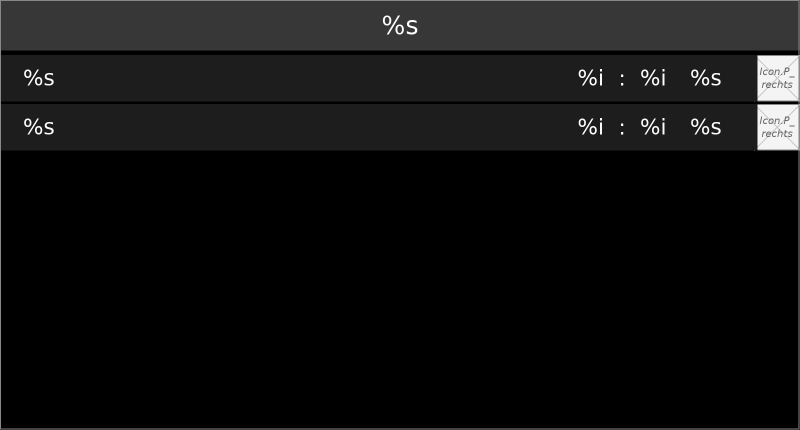
VISUALIZATION CLK_D_Tagesprogramm_Liste  // 800x430
VAR_IN_OUT
	FB_CLK_D:CLK_D;
	
END_VAR
VAR_INPUT
	i_Titel:INT;
END_VAR
	
VAR

	
	
END_VAR
    Rectangle (0,425 800x5)
    Rectangle (0,0 800x50), "%s", text list: 'Sprachen', text index: i_Titel
    Rectangle (0,55 800x46)
    Rectangle (20,55 400x46), "%s", text list: 'Sprachen', text index: 93
    Image (754,55 46x46), image: Icon.P_rechts
        OnMouseClick: execute { Visu.i_Frame_Index:=1; }
    Rectangle (637,55 49x46), "%i", text variable: FB_CLK_D.t_Ein.wMinute
    Rectangle (537,55 70x46), "%i", text variable: FB_CLK_D.t_Ein.wHour
    Rectangle (617,55 10x46), ":"
    Rectangle (687,55 70x46), "%s", text list: 'Sprachen', text index: 74
    Rectangle (0,104 800x46)
    Rectangle (20,104 400x46), "%s", text list: 'Sprachen', text index: 94
    Image (754,104 46x46), image: Icon.P_rechts
        OnMouseClick: execute { Visu.i_Frame_Index:=2; }
    Rectangle (637,104 49x46), "%i", text variable: FB_CLK_D.t_Aus.wMinute
    Rectangle (537,104 70x46), "%i", text variable: FB_CLK_D.t_Aus.wHour
    Rectangle (617,104 10x46), ":"
    Rectangle (687,104 70x46), "%s", text list: 'Sprachen', text index: 74
END_VISUALIZATION

// ZY_Visu/Zeitprogramm/CLK_I/CLK_I_Tagesimpuls
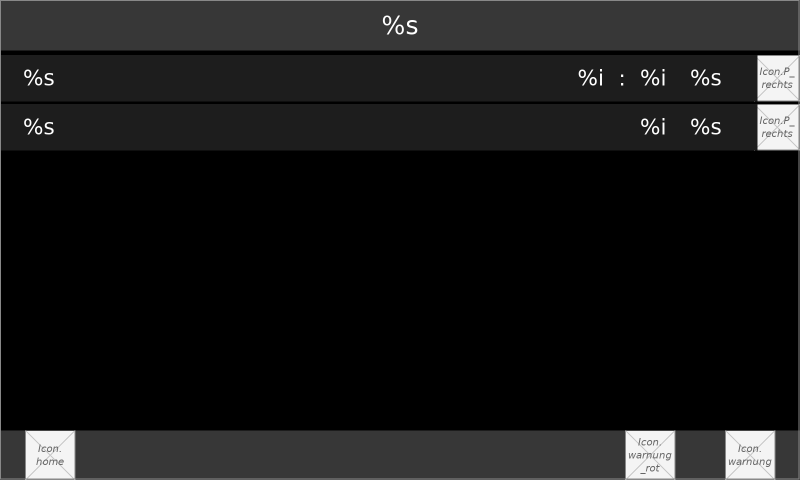
VISUALIZATION CLK_I_Tagesimpuls  // 800x480
VAR_IN_OUT
	FB_CLK_I:CLK_I;

END_VAR
    Frame (0,430 800x50)
        shows Fusszeile_50()
    Frame (0,0 800x430), frame switch variable: Visu.i_Frame_Index
        shows CLK_I_Tagesimpuls_Liste(i_Titel := 76, FB_CLK_I := FB_CLK_I)
        shows Ein_Aus_Zeit_aendern(i_titel := 68, i_Minuten := FB_CLK_I.t_Ein.wMinute, i_Stunden := FB_CLK_I.t_Ein.wHour)
        shows Sekunden_aendern(i_titel := 102, i_Sekunden := FB_CLK_I.t_Imp.wSecond)
END_VISUALIZATION

// ZY_Visu/Zeitprogramm/CLK_I/CLK_I_Tagesimpuls_Liste
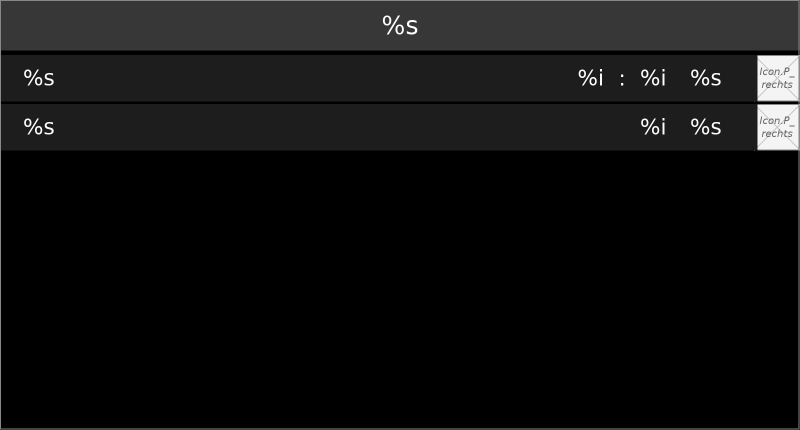
VISUALIZATION CLK_I_Tagesimpuls_Liste  // 800x430
VAR_IN_OUT
	FB_CLK_I:CLK_I;
	
END_VAR
VAR_INPUT
	i_Titel:INT;
END_VAR
	
VAR

	
	
END_VAR
    Rectangle (0,425 800x5)
    Rectangle (0,0 800x50), "%s", text list: 'Sprachen', text index: i_Titel
    Rectangle (0,55 800x46)
    Rectangle (20,55 400x46), "%s", text list: 'Sprachen', text index: 93
    Image (754,55 46x46), image: Icon.P_rechts
        OnMouseClick: execute { Visu.i_Frame_Index:=1; }
    Rectangle (637,55 49x46), "%i", text variable: FB_CLK_I.t_Ein.wMinute
    Rectangle (537,55 70x46), "%i", text variable: FB_CLK_I.t_Ein.wHour
    Rectangle (617,55 10x46), ":"
    Rectangle (687,55 70x46), "%s", text list: 'Sprachen', text index: 74
    Rectangle (0,104 800x46)
    Rectangle (20,104 400x46), "%s", text list: 'Sprachen', text index: 102
    Image (754,104 46x46), image: Icon.P_rechts
        OnMouseClick: execute { Visu.i_Frame_Index:=2; }
    Rectangle (637,104 49x46), "%i", text variable: FB_CLK_I.t_Imp.wSecond
    Rectangle (687,104 70x46), "%s", text list: 'Sprachen', text index: 103
END_VISUALIZATION

// ZY_Visu/Zeitprogramm/CLK_M/CLK_M_Monatsimpuls
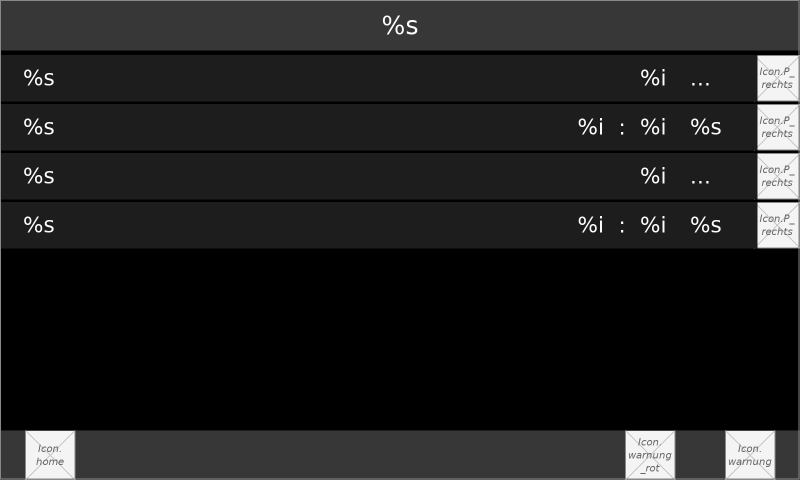
VISUALIZATION CLK_M_Monatsimpuls  // 800x480
VAR_IN_OUT
	FB_CLK_M:CLK_M;

END_VAR
    Frame (0,430 800x50)
        shows Fusszeile_50()
    Frame (0,0 800x430), frame switch variable: Visu.i_Frame_Index
        shows CLK_M_Monatsimpuls_Liste(i_Titel := 78, FB_CLK_M := FB_CLK_M)
        shows Monatstag_aendern(i_titel := 99, i_Monatstag := FB_CLK_M.t_Ein.wDay)
        shows Ein_Aus_Zeit_aendern(i_titel := 68, i_Minuten := FB_CLK_M.t_Ein.wMinute, i_Stunden := FB_CLK_M.t_Ein.wHour)
        shows Monatstag_aendern(i_titel := 99, i_Monatstag := FB_CLK_M.t_Aus.wDay)
        shows Ein_Aus_Zeit_aendern(i_titel := 68, i_Minuten := FB_CLK_M.t_Aus.wMinute, i_Stunden := FB_CLK_M.t_Aus.wHour)
END_VISUALIZATION

// ZY_Visu/Zeitprogramm/CLK_M/CLK_M_Monatsimpuls_Liste
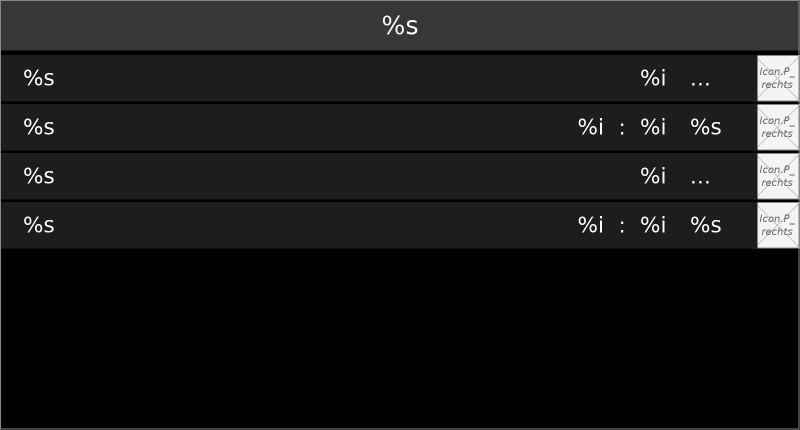
VISUALIZATION CLK_M_Monatsimpuls_Liste  // 800x430
VAR_IN_OUT
	FB_CLK_M:CLK_M;
	
END_VAR
VAR_INPUT
	i_Titel:INT;
END_VAR
	
VAR

	
	
END_VAR
    Rectangle (0,425 800x5)
    Rectangle (0,0 800x50), "%s", text list: 'Sprachen', text index: i_Titel
    Rectangle (0,104 800x46)
    Rectangle (20,104 400x46), "%s", text list: 'Sprachen', text index: 93
    Image (754,104 46x46), image: Icon.P_rechts
        OnMouseClick: execute { Visu.i_Frame_Index:=2; }
    Rectangle (637,104 49x46), "%i", text variable: FB_CLK_M.t_Ein.wMinute
    Rectangle (537,104 70x46), "%i", text variable: FB_CLK_M.t_Ein.wHour
    Rectangle (617,104 10x46), ":"
    Rectangle (687,104 70x46), "%s", text list: 'Sprachen', text index: 74
    Rectangle (0,55 800x46)
    Rectangle (20,55 400x46), "%s", text list: 'Sprachen', text index: 97
    Image (754,55 46x46), image: Icon.P_rechts
        OnMouseClick: execute { Visu.i_Frame_Index:=1; }
    Rectangle (677,55 70x45)
    Rectangle (637,55 49x46), "%i", text variable: FB_CLK_M.t_Ein.wDay
    Rectangle (687,55 70x46), "..."
    Rectangle (0,202 800x46)
    Rectangle (20,202 400x46), "%s", text list: 'Sprachen', text index: 94
    Image (754,202 46x46), image: Icon.P_rechts
        OnMouseClick: execute { Visu.i_Frame_Index:=4; }
    Rectangle (637,202 49x46), "%i", text variable: FB_CLK_M.t_Aus.wMinute
    Rectangle (537,202 70x46), "%i", text variable: FB_CLK_M.t_Aus.wHour
    Rectangle (617,202 10x46), ":"
    Rectangle (687,202 70x46), "%s", text list: 'Sprachen', text index: 74
    Rectangle (0,153 800x46)
    Rectangle (20,153 400x46), "%s", text list: 'Sprachen', text index: 98
    Image (754,153 46x46), image: Icon.P_rechts
        OnMouseClick: execute { Visu.i_Frame_Index:=3; }
    Rectangle (677,153 70x45)
    Rectangle (637,153 49x46), "%i", text variable: FB_CLK_M.t_Aus.wDay
    Rectangle (687,153 70x46), "..."
END_VISUALIZATION

// ZY_Visu/Zeitprogramm/CLK_W/CLK_W_Wochenprogramm
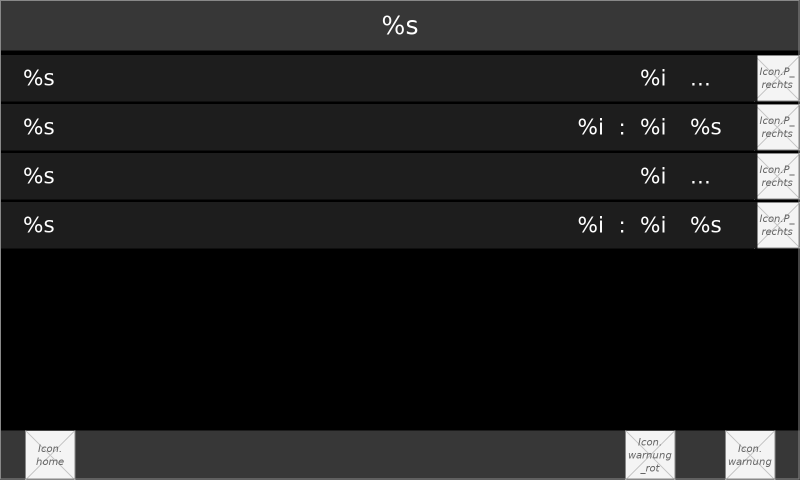
VISUALIZATION CLK_W_Wochenprogramm  // 800x480
VAR_IN_OUT
	FB_CLK_W:CLK_W;

END_VAR
    Frame (0,430 800x50)
        shows Fusszeile_50()
    Frame (0,0 800x430)
        shows CLK_W_Wochenprogramm_Liste(i_Titel := 75, FB_CLK_W := FB_CLK_W)
        shows Wochentag_aendern(i_titel := 80, i_Wochentag := FB_CLK_W.t_Ein.wDayOfWeek)
        shows Ein_Aus_Zeit_aendern(i_titel := 68, i_Minuten := FB_CLK_W.t_Ein.wMinute, i_Stunden := FB_CLK_W.t_Ein.wHour)
        shows Wochentag_aendern(i_titel := 80, i_Wochentag := FB_CLK_W.t_Aus.wDayOfWeek)
        shows Ein_Aus_Zeit_aendern(i_titel := 68, i_Minuten := FB_CLK_W.t_Aus.wMinute, i_Stunden := FB_CLK_W.t_Aus.wHour)
END_VISUALIZATION

// ZY_Visu/Zeitprogramm/CLK_W/CLK_W_Wochenprogramm_Liste
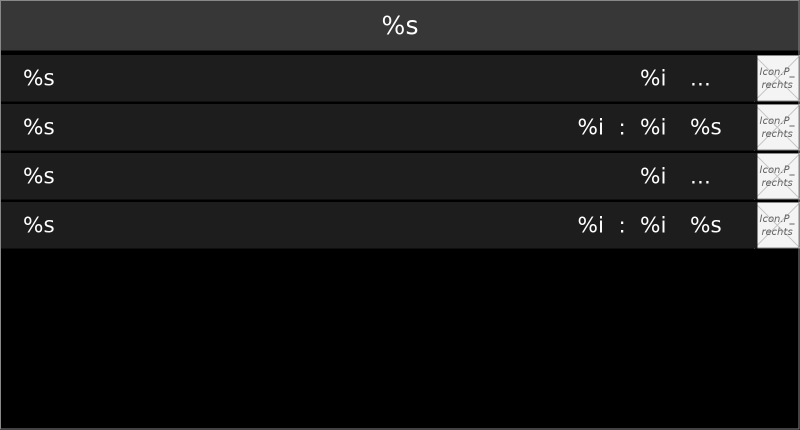
VISUALIZATION CLK_W_Wochenprogramm_Liste  // 800x430
VAR_IN_OUT
	FB_CLK_W:CLK_W;
	
END_VAR
VAR_INPUT
	i_Titel:INT;
END_VAR
	
VAR
	
	
END_VAR
    Rectangle (0,425 800x5)
    Rectangle (0,0 800x50), "%s", text list: 'Sprachen', text index: i_Titel
    Rectangle (0,104 800x46)
    Rectangle (20,104 400x46), "%s", text list: 'Sprachen', text index: 93
    Image (754,104 46x46), image: Icon.P_rechts
        OnMouseClick: execute { Visu.i_Frame_Index:=2; }
    Rectangle (637,104 49x46), "%i", text variable: FB_CLK_W.t_Ein.wMinute
    Rectangle (537,104 70x46), "%i", text variable: FB_CLK_W.t_Ein.wHour
    Rectangle (617,104 10x46), ":"
    Rectangle (687,104 70x46), "%s", text list: 'Sprachen', text index: 74
    Rectangle (0,55 800x46)
    Rectangle (20,55 400x46), "%s", text list: 'Sprachen', text index: 82
    Image (754,55 46x46), image: Icon.P_rechts
        OnMouseClick: execute { Visu.i_Frame_Index:=1; }
    Rectangle (677,55 70x45)
    Rectangle (637,55 49x46), "%i", text variable: FB_CLK_W.t_Ein.wDayOfWeek
    Rectangle (687,55 70x46), "..."
    Rectangle (0,202 800x46)
    Rectangle (20,202 400x46), "%s", text list: 'Sprachen', text index: 94
    Image (754,202 46x46), image: Icon.P_rechts
        OnMouseClick: execute { Visu.i_Frame_Index:=4; }
    Rectangle (637,202 49x46), "%i", text variable: FB_CLK_W.t_Aus.wMinute
    Rectangle (537,202 70x46), "%i", text variable: FB_CLK_W.t_Aus.wHour
    Rectangle (617,202 10x46), ":"
    Rectangle (687,202 70x46), "%s", text list: 'Sprachen', text index: 74
    Rectangle (0,153 800x46)
    Rectangle (20,153 400x46), "%s", text list: 'Sprachen', text index: 83
    Image (754,153 46x46), image: Icon.P_rechts
        OnMouseClick: execute { Visu.i_Frame_Index:=3; }
    Rectangle (677,153 70x45)
    Rectangle (637,153 49x46), "%i", text variable: FB_CLK_W.t_Aus.wDayOfWeek
    Rectangle (687,153 70x46), "..."
END_VISUALIZATION

// ZY_Visu/Zeitprogramm/CLK_W7/CLK_W7_Siebentageprogramm
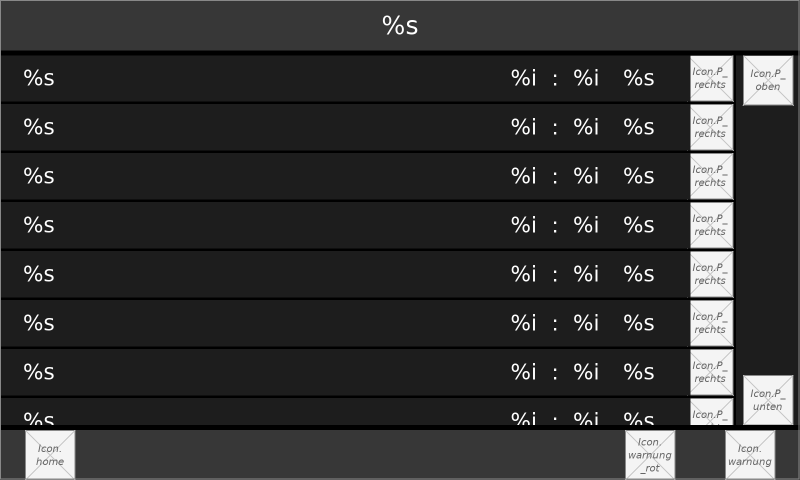
VISUALIZATION CLK_W7_Siebentageprogramm  // 800x480
VAR_IN_OUT
	FB_CLK_W7:CLK_W7;

END_VAR
    Frame (0,0 800x430), frame switch variable: Visu.i_Frame_Index
        shows CLK_W7_Siebentageprogramm_Liste(i_Titel := 95, FB_CLK_W7 := FB_CLK_W7)
        shows Ein_Aus_Zeit_aendern(i_titel := 68, i_Minuten := FB_CLK_W7.t_Ein_Mo.wMinute, i_Stunden := FB_CLK_W7.t_Ein_Mo.wHour)
        shows Ein_Aus_Zeit_aendern(i_titel := 68, i_Minuten := FB_CLK_W7.t_Aus_Mo.wMinute, i_Stunden := FB_CLK_W7.t_Aus_Mo.wHour)
        shows Ein_Aus_Zeit_aendern(i_titel := 68, i_Minuten := FB_CLK_W7.t_Ein_Di.wMinute, i_Stunden := FB_CLK_W7.t_Ein_Di.wHour)
        shows Ein_Aus_Zeit_aendern(i_titel := 68, i_Minuten := FB_CLK_W7.t_Aus_Di.wMinute, i_Stunden := FB_CLK_W7.t_Aus_Di.wHour)
        shows Ein_Aus_Zeit_aendern(i_titel := 68, i_Minuten := FB_CLK_W7.t_Ein_Mi.wMinute, i_Stunden := FB_CLK_W7.t_Ein_Mi.wHour)
        shows Ein_Aus_Zeit_aendern(i_titel := 68, i_Minuten := FB_CLK_W7.t_Aus_Mi.wMinute, i_Stunden := FB_CLK_W7.t_Aus_Mi.wHour)
        shows Ein_Aus_Zeit_aendern(i_titel := 68, i_Minuten := FB_CLK_W7.t_Ein_Do.wMinute, i_Stunden := FB_CLK_W7.t_Ein_Do.wHour)
        shows Ein_Aus_Zeit_aendern(i_titel := 68, i_Minuten := FB_CLK_W7.t_Aus_Do.wMinute, i_Stunden := FB_CLK_W7.t_Aus_Do.wHour)
        shows Ein_Aus_Zeit_aendern(i_titel := 68, i_Minuten := FB_CLK_W7.t_Ein_Fr.wMinute, i_Stunden := FB_CLK_W7.t_Ein_Fr.wHour)
        shows Ein_Aus_Zeit_aendern(i_titel := 68, i_Minuten := FB_CLK_W7.t_Aus_Fr.wMinute, i_Stunden := FB_CLK_W7.t_Aus_Fr.wHour)
        shows Ein_Aus_Zeit_aendern(i_titel := 68, i_Minuten := FB_CLK_W7.t_Ein_Sa.wMinute, i_Stunden := FB_CLK_W7.t_Ein_Sa.wHour)
        shows Ein_Aus_Zeit_aendern(i_titel := 68, i_Minuten := FB_CLK_W7.t_Aus_Sa.wMinute, i_Stunden := FB_CLK_W7.t_Aus_Sa.wHour)
        shows Ein_Aus_Zeit_aendern(i_titel := 68, i_Minuten := FB_CLK_W7.t_Ein_So.wMinute, i_Stunden := FB_CLK_W7.t_Ein_So.wHour)
        shows Ein_Aus_Zeit_aendern(i_titel := 68, i_Minuten := FB_CLK_W7.t_Aus_So.wMinute, i_Stunden := FB_CLK_W7.t_Aus_So.wHour)
    Frame (0,430 800x50)
        shows Fusszeile_50()
END_VISUALIZATION

// ZY_Visu/Zeitprogramm/CLK_W7/CLK_W7_Siebentageprogramm_Liste
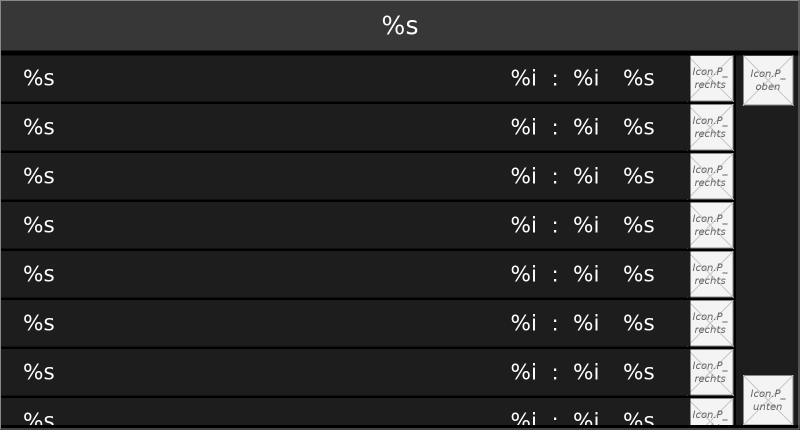
VISUALIZATION CLK_W7_Siebentageprogramm_Liste  // 800x430
VAR_IN_OUT
	FB_CLK_W7:CLK_W7;
	
END_VAR
VAR_INPUT
	i_Titel:INT;
END_VAR
	
VAR
	ton:ton;
	x_ab:BOOL;
	
	
END_VAR
    Group (736,55 64x370)
        Rectangle (0,0 64x370)
        Image (7,320 50x50), image: Icon.P_unten
            OnMouseClick: execute {
                IF  Visu.i_Verschiebung_Vertikal<0 THEN
                Visu.i_Verschiebung_Vertikal:= Visu.i_Verschiebung_Vertikal+52;
                end_if
            }
        Image (7,0 50x50), image: Icon.P_oben
            OnMouseClick: execute {
                IF  Visu.i_Verschiebung_Vertikal>-312 THEN
                Visu.i_Verschiebung_Vertikal:= Visu.i_Verschiebung_Vertikal-52;
                end_if
            }
    Group (0,55 733x683)
        p2738717112: Visu.i_Verschiebung_Vertikal
        Rectangle (0,0 733x46)
        Image (687,0 46x46), image: Icon.P_rechts
            OnMouseClick: execute { Visu.i_Frame_Index:=1; }
        Rectangle (20,0 400x46), "%s", text list: 'Sprachen', text index: 54
        Rectangle (570,0 49x46), "%i", text variable: FB_CLK_W7.t_Ein_Mo.wMinute
        Rectangle (470,0 70x46), "%i", text variable: FB_CLK_W7.t_Ein_Mo.wHour
        Rectangle (550,0 10x46), ":", text variable: FB_CLK_W7.t_Ein_Mo.wMinute
        Rectangle (620,0 70x46), "%s", text list: 'Sprachen', text index: 74
        Rectangle (0,49 733x46)
        Image (687,49 46x46), image: Icon.P_rechts
            OnMouseClick: execute { Visu.i_Frame_Index:=2; }
        Rectangle (610,49 70x45), text variable: FB_CLK_W7.t_Aus_Mo.wMinute
        Rectangle (510,49 70x45), text variable: FB_CLK_W7.t_Aus_Mo.wHour
        Rectangle (20,49 400x46), "%s", text list: 'Sprachen', text index: 55
        Rectangle (570,49 49x46), "%i", text variable: FB_CLK_W7.t_Aus_Mo.wMinute
        Rectangle (470,49 70x46), "%i", text variable: FB_CLK_W7.t_Aus_Mo.wHour
        Rectangle (550,49 10x46), ":", text variable: FB_CLK_W7.t_Ein_Mo.wMinute
        Rectangle (620,49 70x46), "%s", text list: 'Sprachen', text index: 74
        Rectangle (0,98 733x46)
        Image (687,98 46x46), image: Icon.P_rechts
            OnMouseClick: execute { Visu.i_Frame_Index:=3; }
        Rectangle (610,98 70x45), text variable: FB_CLK_W7.t_Aus_Mo.wMinute
        Rectangle (510,98 70x45), text variable: FB_CLK_W7.t_Aus_Mo.wHour
        Rectangle (20,98 400x46), "%s", text list: 'Sprachen', text index: 56
        Rectangle (570,98 49x46), "%i", text variable: FB_CLK_W7.t_Ein_Di.wMinute
        Rectangle (470,98 70x46), "%i", text variable: FB_CLK_W7.t_Ein_Di.wHour
        Rectangle (550,98 10x46), ":", text variable: FB_CLK_W7.t_Ein_Mo.wMinute
        Rectangle (620,98 70x46), "%s", text list: 'Sprachen', text index: 74
        Rectangle (0,147 733x46)
        Image (687,147 46x46), image: Icon.P_rechts
            OnMouseClick: execute { Visu.i_Frame_Index:=4; }
        Rectangle (610,147 70x45), text variable: FB_CLK_W7.t_Aus_Mo.wMinute
        Rectangle (510,147 70x45), text variable: FB_CLK_W7.t_Aus_Mo.wHour
        Rectangle (20,147 400x46), "%s", text list: 'Sprachen', text index: 57
        Rectangle (570,147 49x46), "%i", text variable: FB_CLK_W7.t_Aus_Di.wMinute
        Rectangle (470,147 70x46), "%i", text variable: FB_CLK_W7.t_Aus_Di.wHour
        Rectangle (550,147 10x46), ":", text variable: FB_CLK_W7.t_Ein_Mo.wMinute
        Rectangle (620,147 70x46), "%s", text list: 'Sprachen', text index: 74
        Rectangle (0,196 733x46)
        Image (687,196 46x46), image: Icon.P_rechts
            OnMouseClick: execute { Visu.i_Frame_Index:=5; }
        Rectangle (610,196 70x45), text variable: FB_CLK_W7.t_Aus_Mo.wMinute
        Rectangle (510,196 70x45), text variable: FB_CLK_W7.t_Aus_Mo.wHour
        Rectangle (20,196 400x46), "%s", text list: 'Sprachen', text index: 58
        Rectangle (570,196 49x46), "%i", text variable: FB_CLK_W7.t_Ein_Mi.wMinute
        Rectangle (470,196 70x46), "%i", text variable: FB_CLK_W7.t_Ein_Mi.wHour
        Rectangle (550,196 10x46), ":", text variable: FB_CLK_W7.t_Ein_Mo.wMinute
        Rectangle (620,196 70x46), "%s", text list: 'Sprachen', text index: 74
        Rectangle (0,245 733x46)
        Image (687,245 46x46), image: Icon.P_rechts
            OnMouseClick: execute { Visu.i_Frame_Index:=6; }
        Rectangle (610,245 70x45), text variable: FB_CLK_W7.t_Aus_Mo.wMinute
        Rectangle (510,245 70x45), text variable: FB_CLK_W7.t_Aus_Mo.wHour
        Rectangle (20,245 400x46), "%s", text list: 'Sprachen', text index: 59
        Rectangle (570,245 49x46), "%i", text variable: FB_CLK_W7.t_Aus_Mi.wMinute
        Rectangle (470,245 70x46), "%i", text variable: FB_CLK_W7.t_Aus_Mi.wHour
        Rectangle (550,245 10x46), ":", text variable: FB_CLK_W7.t_Ein_Mo.wMinute
        Rectangle (620,245 70x46), "%s", text list: 'Sprachen', text index: 74
        Rectangle (0,294 733x46)
        Image (687,294 46x46), image: Icon.P_rechts
            OnMouseClick: execute { Visu.i_Frame_Index:=7; }
        Rectangle (610,294 70x45), text variable: FB_CLK_W7.t_Aus_Mo.wMinute
        Rectangle (510,294 70x45), text variable: FB_CLK_W7.t_Aus_Mo.wHour
        Rectangle (20,294 400x46), "%s", text list: 'Sprachen', text index: 60
        Rectangle (570,294 49x46), "%i", text variable: FB_CLK_W7.t_Ein_Do.wMinute
        Rectangle (470,294 70x46), "%i", text variable: FB_CLK_W7.t_Ein_Do.wHour
        Rectangle (550,294 10x46), ":", text variable: FB_CLK_W7.t_Ein_Mo.wMinute
        Rectangle (620,294 70x46), "%s", text list: 'Sprachen', text index: 74
        Rectangle (0,343 733x46)
        Image (687,343 46x46), image: Icon.P_rechts
            OnMouseClick: execute { Visu.i_Frame_Index:=8; }
        Rectangle (610,343 70x45), text variable: FB_CLK_W7.t_Aus_Mo.wMinute
        Rectangle (510,343 70x45), text variable: FB_CLK_W7.t_Aus_Mo.wHour
        Rectangle (20,343 400x46), "%s", text list: 'Sprachen', text index: 61
        Rectangle (570,343 49x46), "%i", text variable: FB_CLK_W7.t_Aus_Do.wMinute
        Rectangle (470,343 70x46), "%i", text variable: FB_CLK_W7.t_Aus_Do.wHour
        Rectangle (550,343 10x46), ":", text variable: FB_CLK_W7.t_Ein_Mo.wMinute
        Rectangle (620,343 70x46), "%s", text list: 'Sprachen', text index: 74
        Rectangle (0,392 733x46)
        Image (687,392 46x46), image: Icon.P_rechts
            OnMouseClick: execute { Visu.i_Frame_Index:=9; }
        Rectangle (20,392 400x46), "%s", text list: 'Sprachen', text index: 62
        Rectangle (570,392 49x46), "%i", text variable: FB_CLK_W7.t_Ein_Fr.wMinute
        Rectangle (470,392 70x46), "%i", text variable: FB_CLK_W7.t_Ein_Fr.wHour
        Rectangle (550,392 10x46), ":", text variable: FB_CLK_W7.t_Ein_Mo.wMinute
        Rectangle (620,392 70x46), "%s", text list: 'Sprachen', text index: 74
        Rectangle (0,490 733x46)
        Image (687,490 46x46), image: Icon.P_rechts
            OnMouseClick: execute { Visu.i_Frame_Index:=11; }
        Rectangle (610,490 70x45), text variable: FB_CLK_W7.t_Aus_Mo.wMinute
        Rectangle (510,490 70x45), text variable: FB_CLK_W7.t_Aus_Mo.wHour
        Rectangle (20,490 400x46), "%s", text list: 'Sprachen', text index: 64
        Rectangle (570,490 49x46), "%i", text variable: FB_CLK_W7.t_Ein_Sa.wMinute
        Rectangle (470,490 70x46), "%i", text variable: FB_CLK_W7.t_Ein_Sa.wHour
        Rectangle (550,490 10x46), ":", text variable: FB_CLK_W7.t_Ein_Mo.wMinute
        Rectangle (620,490 70x46), "%s", text list: 'Sprachen', text index: 74
        Rectangle (0,539 733x46)
        Image (687,539 46x46), image: Icon.P_rechts
            OnMouseClick: execute { Visu.i_Frame_Index:=12; }
        Rectangle (610,539 70x45), text variable: FB_CLK_W7.t_Aus_Mo.wMinute
        Rectangle (510,539 70x45), text variable: FB_CLK_W7.t_Aus_Mo.wHour
        Rectangle (20,539 400x46), "%s", text list: 'Sprachen', text index: 65
        Rectangle (570,539 49x46), "%i", text variable: FB_CLK_W7.t_Aus_Sa.wMinute
        Rectangle (470,539 70x46), "%i", text variable: FB_CLK_W7.t_Aus_Sa.wHour
        Rectangle (550,539 10x46), ":", text variable: FB_CLK_W7.t_Ein_Mo.wMinute
        Rectangle (620,539 70x46), "%s", text list: 'Sprachen', text index: 74
        Rectangle (0,588 733x46)
        Image (687,588 46x46), image: Icon.P_rechts
            OnMouseClick: execute { Visu.i_Frame_Index:=13; }
        Rectangle (610,588 70x45), text variable: FB_CLK_W7.t_Aus_Mo.wMinute
        Rectangle (510,588 70x45), text variable: FB_CLK_W7.t_Aus_Mo.wHour
        Rectangle (20,588 400x46), "%s", text list: 'Sprachen', text index: 66
        Rectangle (570,588 49x46), "%i", text variable: FB_CLK_W7.t_Ein_So.wMinute
        Rectangle (470,588 70x46), "%i", text variable: FB_CLK_W7.t_Ein_So.wHour
        Rectangle (550,588 10x46), ":", text variable: FB_CLK_W7.t_Ein_Mo.wMinute
        Rectangle (620,588 70x46), "%s", text list: 'Sprachen', text index: 74
        Rectangle (0,637 733x46)
        Image (687,637 46x46), image: Icon.P_rechts
            OnMouseClick: execute { Visu.i_Frame_Index:=14; }
        Rectangle (610,637 70x45), text variable: FB_CLK_W7.t_Aus_Mo.wMinute
        Rectangle (510,637 70x45), text variable: FB_CLK_W7.t_Aus_Mo.wHour
        Rectangle (20,637 400x46), "%s", text list: 'Sprachen', text index: 67
        Rectangle (570,637 49x46), "%i", text variable: FB_CLK_W7.t_Aus_So.wMinute
        Rectangle (470,637 70x46), "%i", text variable: FB_CLK_W7.t_Aus_So.wHour
        Rectangle (550,637 10x46), ":", text variable: FB_CLK_W7.t_Ein_Mo.wMinute
        Rectangle (620,637 70x46), "%s", text list: 'Sprachen', text index: 74
        Rectangle (0,441 733x46)
        Image (687,441 46x46), image: Icon.P_rechts
            OnMouseClick: execute { Visu.i_Frame_Index:=10; }
        Rectangle (20,441 400x46), "%s", text list: 'Sprachen', text index: 63
        Rectangle (570,441 49x46), "%i", text variable: FB_CLK_W7.t_Aus_Fr.wMinute
        Rectangle (470,441 70x46), "%i", text variable: FB_CLK_W7.t_Aus_Fr.wHour
        Rectangle (550,441 10x46), ":", text variable: FB_CLK_W7.t_Ein_Mo.wMinute
        Rectangle (620,441 70x46), "%s", text list: 'Sprachen', text index: 74
    Rectangle (0,50 800x5)
    Rectangle (0,425 800x5)
    Rectangle (0,0 800x50), "%s", text list: 'Sprachen', text index: i_Titel
END_VISUALIZATION

(* text list Alarme (id | default | Deutsch)
  0 | ID0 | 
  1 | ID1 | 
  2 | ID2 | 
  3 | ID3 | 
  4 | ID4 | 
  5 | ID5 | 
  6 | ID6 | 
  7 | ID7 | 
  8 | ID8 | 
  9 | ID9 | 
  10 | ID10 | 
  11 | ID11 | 
  12 | ID12 | 
  13 | ID13 | 
  14 | ID14 | 
  15 | ID15 | 
  16 | ID16 | 
  17 | ID17 | 
  18 | ID18 | 
  19 | ID19 | 
  20 | ID20 | 
  21 | ID21 | 
  22 | ID22 | 
  23 | ID23 | 
  24 | ID24 | 
  25 | ID25 | 
  26 | ID26 | 
  27 | ID27 | 
  28 | ID28 | 
  29 | ID29 | 
  30 | ID30 | 
  31 | ID31 | 
  32 | ID32 | 
  33 | ID33 | 
  34 | ID34 | 
  35 | ID35 | 
  36 | ID36 | 
  37 | ID37 | 
  38 | ID38 | 
  39 | ID39 | 
  40 | ID40 | 
  41 | ID41 | 
  42 | ID42 | 
  43 | ID43 | 
  44 | ID44 | 
  45 | ID45 | 
  46 | ID46 | 
  47 | ID47 | 
  48 | ID48 | 
  49 | ID49 | 
  50 | ID50 | 
  51 | ID51 | 
  52 | ID52 | 
  53 | ID53 | 
  54 | ID54 | 
  55 | ID55 | 
  56 | ID56 | 
  57 | ID57 | 
  58 | ID58 | 
  59 | ID59 | 
  60 | ID60 | 
  61 | ID61 | 
  62 | ID62 | 
  63 | ID63 | 
  64 | ID64 | 
  65 | ID65 | 
  66 | ID66 | 
  67 | ID67 | 
  68 | ID68 | 
  69 | ID69 | 
  70 | ID70 | 
  71 | ID71 | 
  72 | ID72 | 
  73 | ID73 | 
  74 | ID74 | 
  75 | ID75 | 
  76 | ID76 | 
  77 | ID77 | 
  78 | ID78 | 
  79 | ID79 | 
  80 | ID80 | 
  81 | ID81 | 
  82 | ID82 | 
  83 | ID83 | 
  84 | ID84 | 
  85 | ID85 | 
  86 | ID86 | 
  87 | ID87 | 
  88 | ID88 | 
  89 | ID89 | 
  90 | ID90 | 
  91 | ID91 | 
  92 | ID92 | 
  93 | ID93 | 
  94 | ID94 | 
  95 | ID95 | 
  96 | ID96 | 
  97 | ID97 | 
  98 | ID98 | 
  99 | ID99 | 
   |  |  *)

(* text list Sprachen (id | default | Deutsch | Englisch | De)
  100 | Verzoegerung Stufe 2 |  |  | 
  101 | Verzögerung Stufe 1 |  |  | 
  0 | Wärmegewinnung |  |  | 
  1 | Wärmepumpe |  |  | 
  2 | Wärmesenke |  |  | 
  3 | Sollwertmenue |  |  | 
  4 | Sollwerte Wärmegewinnung |  |  | 
  5 | UWP Verd. |  |  | 
  6 | Erdsonde |  |  | 
  7 | Grundwasser |  |  | 
  8 | Luft |  |  | 
  9 | Tiefhaltung |  |  | 
  10 | Abtauspeicher |  |  | 
  11 | Abtauungen |  |  | 
  12 | Abwärme |  |  | 
  13 |  |  |  | 
  14 | Sollwerte Wärmepumpe |  |  | 
  15 | EEV |  |  | 
  16 | Einsatzgrenzen |  |  | 
  17 | Verdichter |  |  | 
  18 | Allgemein |  |  | 
  19 | Sollwerte Wärmesenke |  |  | 
  20 | UWP Verflüssiger |  |  | 
  21 | HWP |  |  | 
  22 | TWW |  |  | 
  23 | Heizgruppe |  |  | 
  24 | Hochhaltung |  |  | 
  25 | Sollwerte UWP Verflüssiger |  |  | 
  26 | Sollwerte Erdsonden |  |  | 
  27 | Sollwerte Luft |  |  | 
  28 | Sollwerte Abwärme |  |  | 
  29 | Sollwerte Tiefhaltung |  |  | 
  30 | Sollwertänderung  |  |  | 
  31 | Infoseite |  |  | 
  32 | Hauptmenü |  |  | 
  33 | Sprachen |  |  | 
  34 | Login |  |  | 
  35 | Sollwerte |  |  | 
  36 | Verlaufs- diagramm |  |  | 
  37 | Uhrzeit einstellen |  |  | 
  38 | IBN |  |  | 
  39 | Konfiguration |  |  | 
  40 | Kontakt |  |  | 
  41 | Ein/Aus Wärmepumpe |  |  | 
  42 | Ein |  |  | 
  43 | Aus |  |  | 
  44 | IO-Auswahl |  |  | 
  45 | Digitale Eingänge |  |  | 
  46 | Digitale Ausgänge |  |  | 
  47 | Analoge Eingänge |  |  | 
  48 | Analoge Ausgänge |  |  | 
  49 | Status |  |  | 
  50 | Offset |  |  | 
  51 | Istwert |  |  | 
  52 | 7 Tage Programm |  |  | 
  53 | Start Zeit |  |  | 
  5000 | Alarme |  |  | 
  54 | Montag Ein |  |  | 
  55 | Montag Aus |  |  | 
  56 | Dienstag Ein |  |  | 
  57 | Dienstag Aus |  |  | 
  58 | Mittwoch Ein |  |  | 
  59 | Mittwoch Aus |  |  | 
  60 | Donnerstag Ein |  |  | 
  61 | Donnerstag Aus |  |  | 
  62 | Freitag Ein |  |  | 
  63 | Freitag Aus |  |  | 
  64 | Samstag Ein |  |  | 
  65 | Samstag Aus |  |  | 
  66 | Sonntag Ein |  |  | 
  67 | Sonntag Aus |  |  | 
  68 | Ein-/Ausschaltzeit  |  |  | 
  69 | Sollwertänderung |  |  | 
  70 | Sprach Auswahl |  |  | 
  71 | Heizkurve |  |  | 
  84 | Dynamischer MOP |  |  | 
  85 | Sollwert Überhitzung |  |  | 
  86 | Maximaler Operating Pressure |  |  | 
  87 | P-Faktor für Regelung |  |  | 
  88 | I-Faktor für Regelung |  |  | 
  89 | D-Faktor für Regelung |  |  | 
  90 | Berechnungstakt PID Regler |  |  | 
  91 | Minimale Überhitzung |  |  | 
  92 | Zeit bis Alarm ausgelöst wird |  |  | 
  96 | Sollwerte EEV |  |  | 
  73 | Abbrechen |  |  | 
  72 | Sollwerte zurücksetzen |  |  | 
  74 | Uhr |  |  | 
  75 | Wochenprogramm |  |  | 
  76 | Tagesimpuls |  |  | 
  77 | Tagesprogramm |  |  | 
  78 | Monatsimpuls |  |  | 
  79 | Jahresprogramm |  |  | 
  80 | Wochentag |  |  | 
  81 | Monat |  |  | 
  82 | Ein Wochentag  |  |  | 
  83 | Aus Wochentag  |  |  | 
  93 | Einschaltzeit |  |  | 
  94 | Ausschaltzeit |  |  | 
  95 | 7 Tage Programm |  |  | 
  97 | Ein Monatstag |  |  | 
  98 | Aus Monatstag |  |  | 
  99 | Monatstag |  |  | 
  102 | Impulsdauer |  |  | 
  103 | Sek |  |  | 
  104 | Ein Monat |  |  | 
  105 | Aus Monat |  |  | 
  106 | Freigabe Heizen |  |  | 
  107 | Tag-/Nachtakivierung |  |  | 
  108 | Aussentemperatur |  |  | 
  109 | Berechnete Aussentemperatur |  |  | 
  110 |  |  |  | 
   |  |  |  |  *)
